{attribute 'qualified_only'}
{attribute 'strict'}
TYPE E_OperatingMode_EMS :
(
	eAllOff := 0,					//{#lynus.ag#()}
	eSelfConsumption := 1,
	ePeakLoadCapping := 2,
	eLoadManagement := 3
);
END_TYPE

(* stored: Version 1.1.0.1, ProductVersion 3.1.4024.9
   DUT E_OperatingMode_EMS: Id {54bcdd33-748a-4a2e-bdaa-1e9ac5811608} *)
